Staubli VAL3: MoveIdWatchdog.pgx

public program moveIdWatchdog()
  local bool l_bLoop
  local num l_nCurrMoveId
  local num l_nIndex
  local num l_nLastMoveId
  local string l_sTemp
  local bool l_bStackWasPop
begin

  //this program run as task can detect moveId alteration...sure there must be a better way to do it...
  //note:
  //      - it doesn't detect a setMoveId if it cause a moveId change < = 1
  //      - is done this way and not on the mere difference beacuse for some reason, sometime the moveId seems having a +-1 discontinuity for a single cicle...
  //        (see SRC-893)

  l_nLastMoveId=getMoveId()
  l_bLoop=true

  while l_bLoop

    l_nCurrMoveId=getMoveId()

    if (roundDown(l_nCurrMoveId)>roundDown(l_nLastMoveId)+1) or (roundDown(l_nCurrMoveId)<roundDown(l_nLastMoveId)-1) or (l_bStackWasPop and isEmpty())
      //resetMotion or SetMoveId detected!
      logMsg("libSignals/moveIdWatchdog->resetMotion or SetMoveId detected")
      setMutex(bAdvMoves)
      call destroyAdvMoves()
      bAdvMoves=false
    endIf

    l_nLastMoveId=l_nCurrMoveId
    //save if the movement stack was populated
    l_bStackWasPop=!isEmpty()

    //if possible kill the moveid watchdog task
    l_bLoop=false
    for l_nIndex=0 to size(bAdvMoveBusy)-1
      l_bLoop=l_bLoop or bAdvMoveBusy[l_nIndex]
    endFor

    delay(0)
  endWhile

end
